(*
A broadcastable wrapper for a `BOOL` value. 
*)
INTERFACE I_BoolArg EXTENDS I_Arg

(*
Reads the internal value.
*)
PROPERTY Get : BOOL
GET
END_GET
END_PROPERTY

(*
Returns TRUE if the value is mutable.
*)
PROPERTY IsMut : BOOL
GET
END_GET
END_PROPERTY

(*
Modifies the internal value.  
Returns:
- `Ok` - Upon successful modification.
- `Error` - If mutability is disabled.
*)
METHOD Set : Result
VAR_INPUT
	newVal		: BOOL;
END_VAR
END_METHOD

END_INTERFACE

(* stored: Version 1.1.0.1
   Itf I_BoolArg: Id {9d76ad8d-669f-4c52-a5c1-5fd937e33189}
   Property Get: Id {d360dbc3-a5ed-481e-8c7d-c7681ec76bb3}
   Get Get: Id {87bd3174-4297-4274-af27-33921f8ed0eb}
   Property IsMut: Id {73297ce6-4a2f-4ad6-9d7a-082014973c25}
   Get Get: Id {0da03f46-1e1d-4476-a665-eabaeee1e20c}
   Method Set: Id {f8bd1ee5-5e13-4cfa-9bd9-124641f0eed9} *)
